(* CoDeSys 2.3 export: PRG_MOVETODEST.EXP *)

(* POU Processes/PRG_MoveToDest, SFC *)
PROGRAM PRG_MoveToDest
VAR_INPUT
	bExecute: BOOL;
	wTarget : WORD;
END_VAR
VAR_INPUT
	bDone: BOOL;
END_VAR
VAR
	tonMoveDelay	: TON;
	tonEjectDelay	: TON;
	tonSensorDelay	: TON;
	tMoveDelay		: TIME := T#500ms;
	tEjectorDelay	: TIME := T#1s;
	tSensorDelay	: TIME := T#500ms;
END_VAR
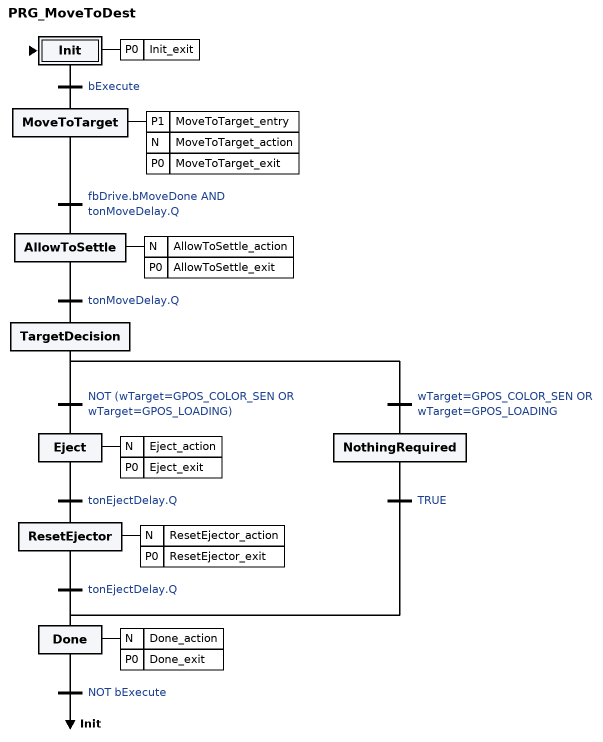
INITIAL_STEP Init:
	Init_exit(P0);
END_STEP
TRANSITION FROM Init TO MoveToTarget := bExecute;
END_TRANSITION
STEP MoveToTarget:
	MoveToTarget_entry(P1);
	MoveToTarget_action(N);
	MoveToTarget_exit(P0);
END_STEP
TRANSITION FROM MoveToTarget TO AllowToSettle := fbDrive.bMoveDone AND tonMoveDelay.Q;
END_TRANSITION
STEP AllowToSettle:
	AllowToSettle_action(N);
	AllowToSettle_exit(P0);
END_STEP
TRANSITION FROM AllowToSettle TO TargetDecision := tonMoveDelay.Q;
END_TRANSITION
STEP TargetDecision:
END_STEP
TRANSITION FROM TargetDecision TO Eject := NOT (wTarget=GPOS_COLOR_SEN OR wTarget=GPOS_LOADING);
END_TRANSITION
TRANSITION FROM TargetDecision TO NothingRequired := wTarget=GPOS_COLOR_SEN OR wTarget=GPOS_LOADING;
END_TRANSITION
STEP NothingRequired:
END_STEP
TRANSITION FROM NothingRequired TO Done := TRUE;
END_TRANSITION
STEP Eject:
	Eject_action(N);
	Eject_exit(P0);
END_STEP
TRANSITION FROM Eject TO ResetEjector := tonEjectDelay.Q;
END_TRANSITION
STEP ResetEjector:
	ResetEjector_action(N);
	ResetEjector_exit(P0);
END_STEP
TRANSITION FROM ResetEjector TO Done := tonEjectDelay.Q;
END_TRANSITION
STEP Done:
	Done_action(N);
	Done_exit(P0);
END_STEP
TRANSITION FROM Done TO Init := NOT bExecute;
END_TRANSITION

ACTION Init_exit:
bDone := FALSE;
END_ACTION

ACTION MoveToTarget_entry:
tonMoveDelay(IN:=FALSE);
END_ACTION

ACTION MoveToTarget_action:
(*Drive Move Delay *)
tonMoveDelay(IN:=TRUE, PT:= T_DRIVE_DELAY);
(* Drive To Target *)
fbDrive(
	bEnable:= TRUE,
	bStart:= TRUE,
	wTarget:= wTarget);
END_ACTION

ACTION MoveToTarget_exit:
fbDrive(
	bStart:= FALSE);
tonMoveDelay(IN:=FALSE);
END_ACTION

ACTION AllowToSettle_action:
tonMoveDelay(IN:=TRUE , PT:= T_POS_SETTLE_DELAY);
END_ACTION

ACTION AllowToSettle_exit:
tonMoveDelay(IN:=FALSE);
END_ACTION

ACTION Eject_action:
tonEjectDelay(IN:=TRUE , PT:= T_EJECTOR_DELAY);
OEjector := TRUE;
END_ACTION

ACTION Eject_exit:
tonEjectDelay(IN:=FALSE);
END_ACTION

ACTION ResetEjector_action:
(* Retract Ejector *)
tonEjectDelay(IN:=TRUE , PT:= T_EJECTOR_DELAY);
OEjector := FALSE;
END_ACTION

ACTION ResetEjector_exit:
tonEjectDelay(IN:=FALSE);
END_ACTION

ACTION Done_action:
bDone := TRUE;
END_ACTION

ACTION Done_exit:
bDone := FALSE;
END_ACTION
END_PROGRAM
